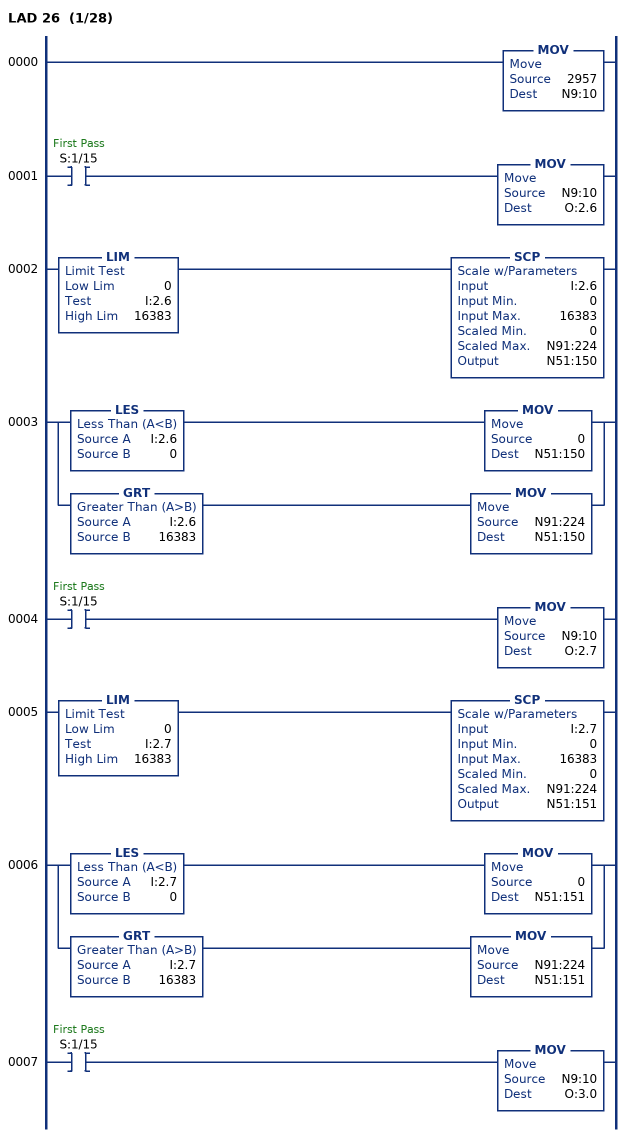
% Rung: 0 %
SOR MOV 2957 N9:10 EOR
% Rung: 1 %
SOR XIC S:1/15 MOV N9:10 O:2.6 EOR
%   S:1/15  "First Pass" %
% Rung: 2 %
SOR LIM 0 I:2.6 16383 SCP I:2.6 0 16383 0 N91:224 N51:150 EOR
% Rung: 3 %
SOR BST LES I:2.6 0 MOV 0 N51:150 NXB GRT I:2.6 16383 MOV N91:224 N51:150 BND EOR
% Rung: 4 %
SOR XIC S:1/15 MOV N9:10 O:2.7 EOR
%   S:1/15  "First Pass" %
% Rung: 5 %
SOR LIM 0 I:2.7 16383 SCP I:2.7 0 16383 0 N91:224 N51:151 EOR
% Rung: 6 %
SOR BST LES I:2.7 0 MOV 0 N51:151 NXB GRT I:2.7 16383 MOV N91:224 N51:151 BND EOR
% Rung: 7 %
SOR XIC S:1/15 MOV N9:10 O:3.0 EOR
%   S:1/15  "First Pass" %

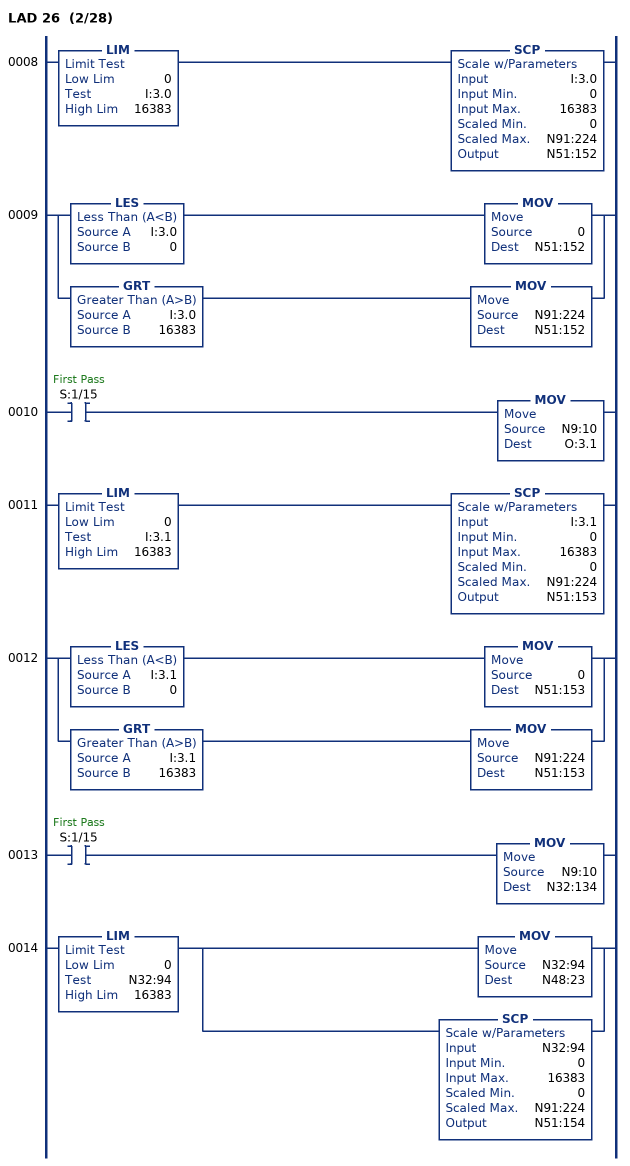
% Rung: 8 %
SOR LIM 0 I:3.0 16383 SCP I:3.0 0 16383 0 N91:224 N51:152 EOR
% Rung: 9 %
SOR BST LES I:3.0 0 MOV 0 N51:152 NXB GRT I:3.0 16383 MOV N91:224 N51:152 BND EOR
% Rung: 10 %
SOR XIC S:1/15 MOV N9:10 O:3.1 EOR
%   S:1/15  "First Pass" %
% Rung: 11 %
SOR LIM 0 I:3.1 16383 SCP I:3.1 0 16383 0 N91:224 N51:153 EOR
% Rung: 12 %
SOR BST LES I:3.1 0 MOV 0 N51:153 NXB GRT I:3.1 16383 MOV N91:224 N51:153 BND EOR
% Rung: 13 %
SOR XIC S:1/15 MOV N9:10 N32:134 EOR
%   S:1/15  "First Pass" %
% Rung: 14 %
SOR LIM 0 N32:94 16383 BST MOV N32:94 N48:23 NXB SCP N32:94 0 16383 0 N91:224 N51:154 BND EOR

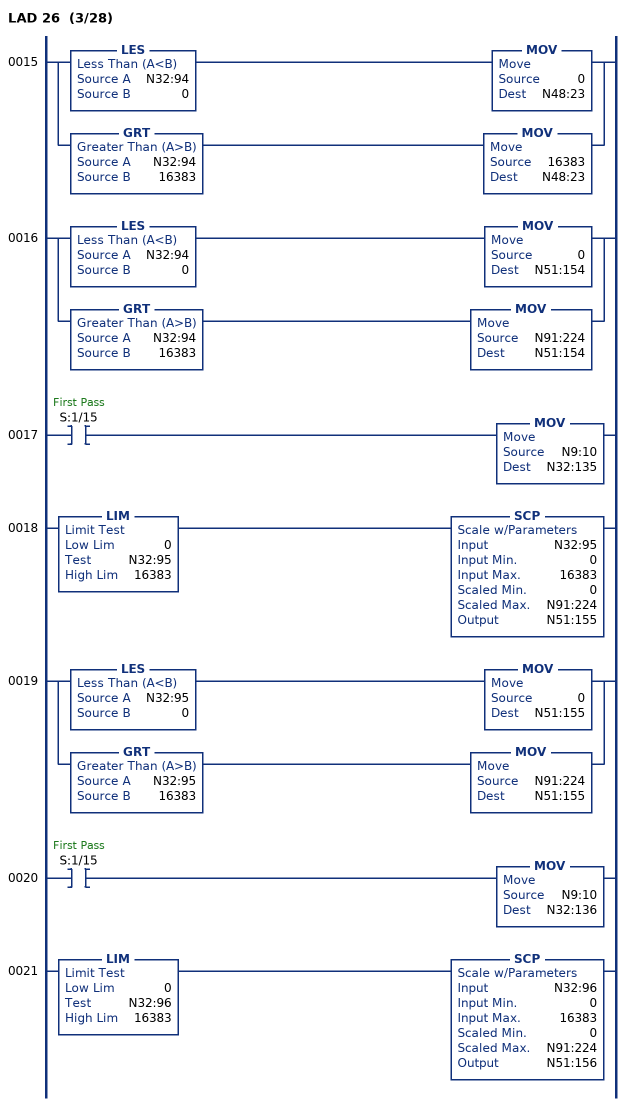
% Rung: 15 %
SOR BST LES N32:94 0 MOV 0 N48:23 NXB GRT N32:94 16383 MOV 16383 N48:23 BND EOR
% Rung: 16 %
SOR BST LES N32:94 0 MOV 0 N51:154 NXB GRT N32:94 16383 MOV N91:224 N51:154 BND EOR
% Rung: 17 %
SOR XIC S:1/15 MOV N9:10 N32:135 EOR
%   S:1/15  "First Pass" %
% Rung: 18 %
SOR LIM 0 N32:95 16383 SCP N32:95 0 16383 0 N91:224 N51:155 EOR
% Rung: 19 %
SOR BST LES N32:95 0 MOV 0 N51:155 NXB GRT N32:95 16383 MOV N91:224 N51:155 BND EOR
% Rung: 20 %
SOR XIC S:1/15 MOV N9:10 N32:136 EOR
%   S:1/15  "First Pass" %
% Rung: 21 %
SOR LIM 0 N32:96 16383 SCP N32:96 0 16383 0 N91:224 N51:156 EOR

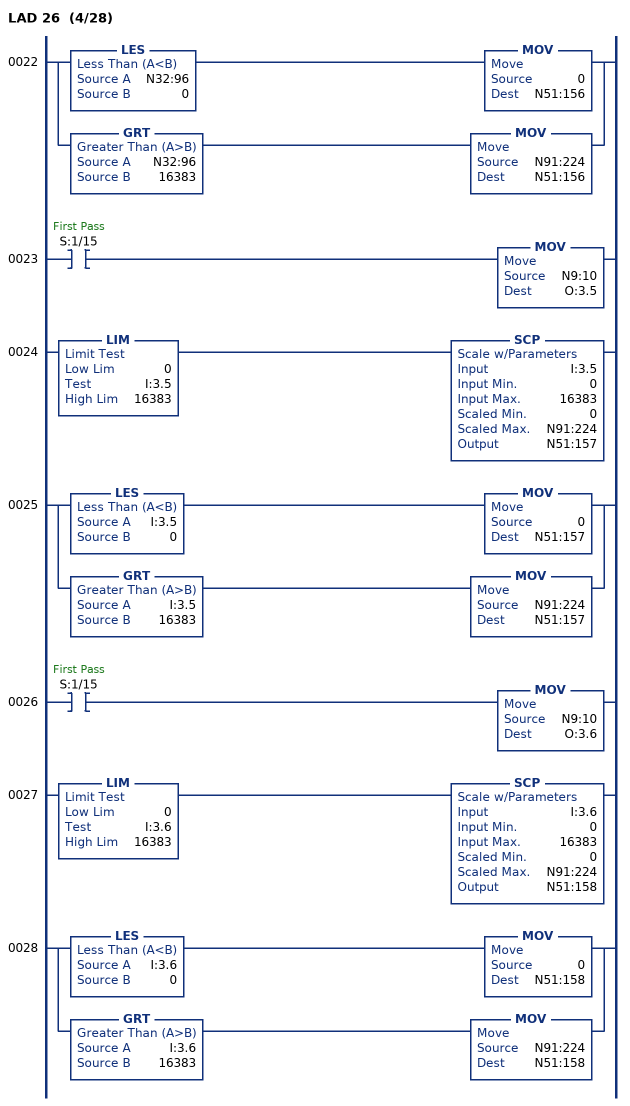
% Rung: 22 %
SOR BST LES N32:96 0 MOV 0 N51:156 NXB GRT N32:96 16383 MOV N91:224 N51:156 BND EOR
% Rung: 23 %
SOR XIC S:1/15 MOV N9:10 O:3.5 EOR
%   S:1/15  "First Pass" %
% Rung: 24 %
SOR LIM 0 I:3.5 16383 SCP I:3.5 0 16383 0 N91:224 N51:157 EOR
% Rung: 25 %
SOR BST LES I:3.5 0 MOV 0 N51:157 NXB GRT I:3.5 16383 MOV N91:224 N51:157 BND EOR
% Rung: 26 %
SOR XIC S:1/15 MOV N9:10 O:3.6 EOR
%   S:1/15  "First Pass" %
% Rung: 27 %
SOR LIM 0 I:3.6 16383 SCP I:3.6 0 16383 0 N91:224 N51:158 EOR
% Rung: 28 %
SOR BST LES I:3.6 0 MOV 0 N51:158 NXB GRT I:3.6 16383 MOV N91:224 N51:158 BND EOR

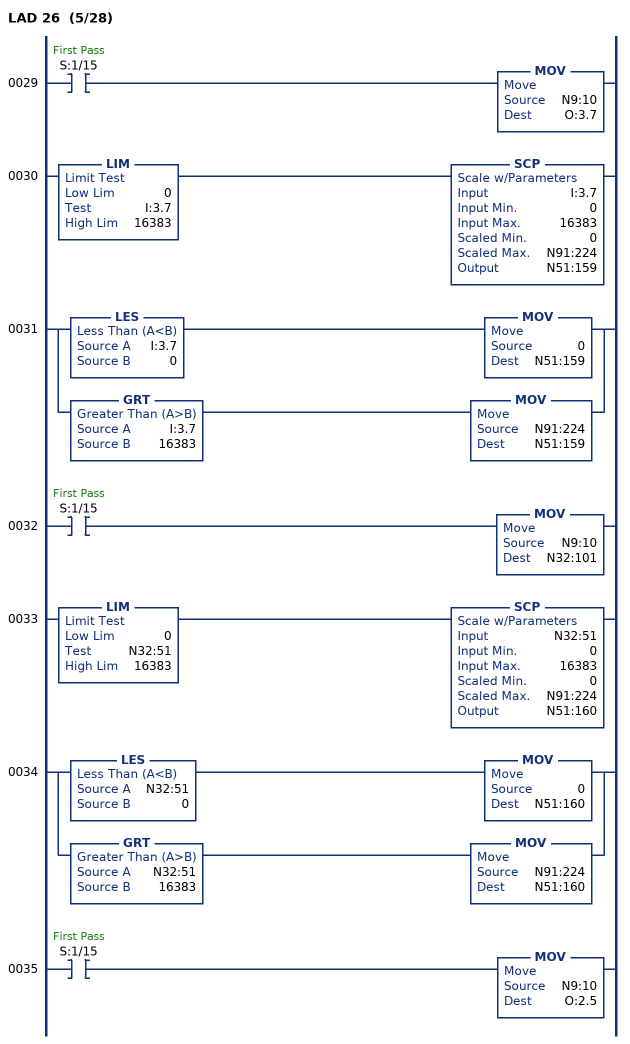
% Rung: 29 %
SOR XIC S:1/15 MOV N9:10 O:3.7 EOR
%   S:1/15  "First Pass" %
% Rung: 30 %
SOR LIM 0 I:3.7 16383 SCP I:3.7 0 16383 0 N91:224 N51:159 EOR
% Rung: 31 %
SOR BST LES I:3.7 0 MOV 0 N51:159 NXB GRT I:3.7 16383 MOV N91:224 N51:159 BND EOR
% Rung: 32 %
SOR XIC S:1/15 MOV N9:10 N32:101 EOR
%   S:1/15  "First Pass" %
% Rung: 33 %
SOR LIM 0 N32:51 16383 SCP N32:51 0 16383 0 N91:224 N51:160 EOR
% Rung: 34 %
SOR BST LES N32:51 0 MOV 0 N51:160 NXB GRT N32:51 16383 MOV N91:224 N51:160 BND EOR
% Rung: 35 %
SOR XIC S:1/15 MOV N9:10 O:2.5 EOR
%   S:1/15  "First Pass" %

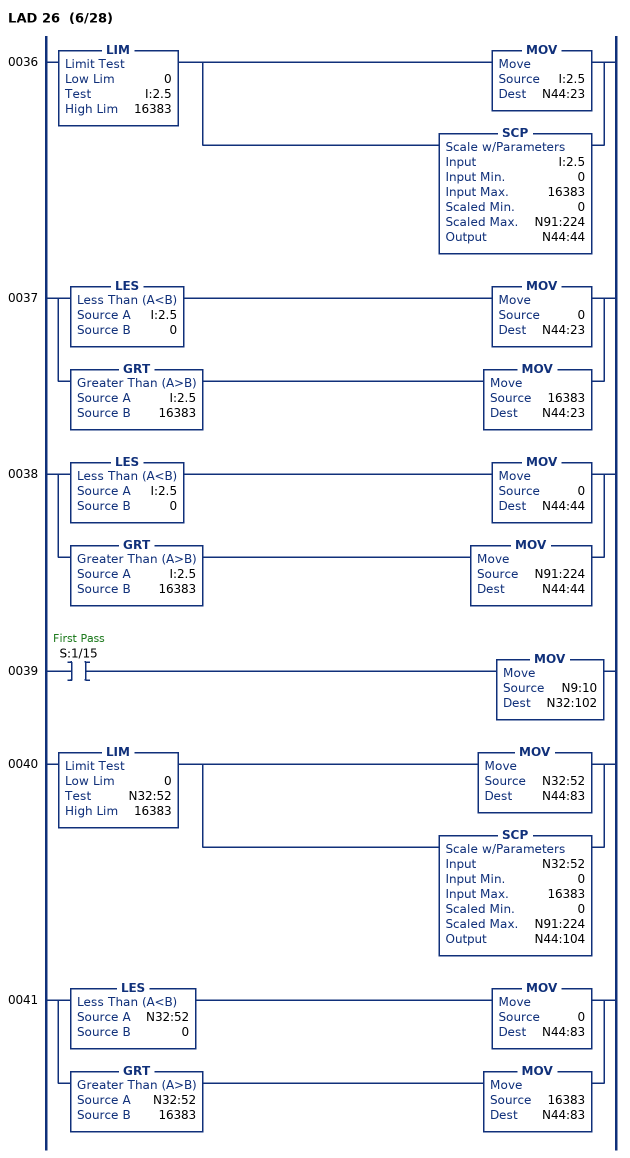
% Rung: 36 %
SOR LIM 0 I:2.5 16383 BST MOV I:2.5 N44:23 NXB SCP I:2.5 0 16383 0 N91:224 N44:44 BND EOR
% Rung: 37 %
SOR BST LES I:2.5 0 MOV 0 N44:23 NXB GRT I:2.5 16383 MOV 16383 N44:23 BND EOR
% Rung: 38 %
SOR BST LES I:2.5 0 MOV 0 N44:44 NXB GRT I:2.5 16383 MOV N91:224 N44:44 BND EOR
% Rung: 39 %
SOR XIC S:1/15 MOV N9:10 N32:102 EOR
%   S:1/15  "First Pass" %
% Rung: 40 %
SOR LIM 0 N32:52 16383 BST MOV N32:52 N44:83 NXB SCP N32:52 0 16383 0 N91:224 N44:104 BND EOR
% Rung: 41 %
SOR BST LES N32:52 0 MOV 0 N44:83 NXB GRT N32:52 16383 MOV 16383 N44:83 BND EOR

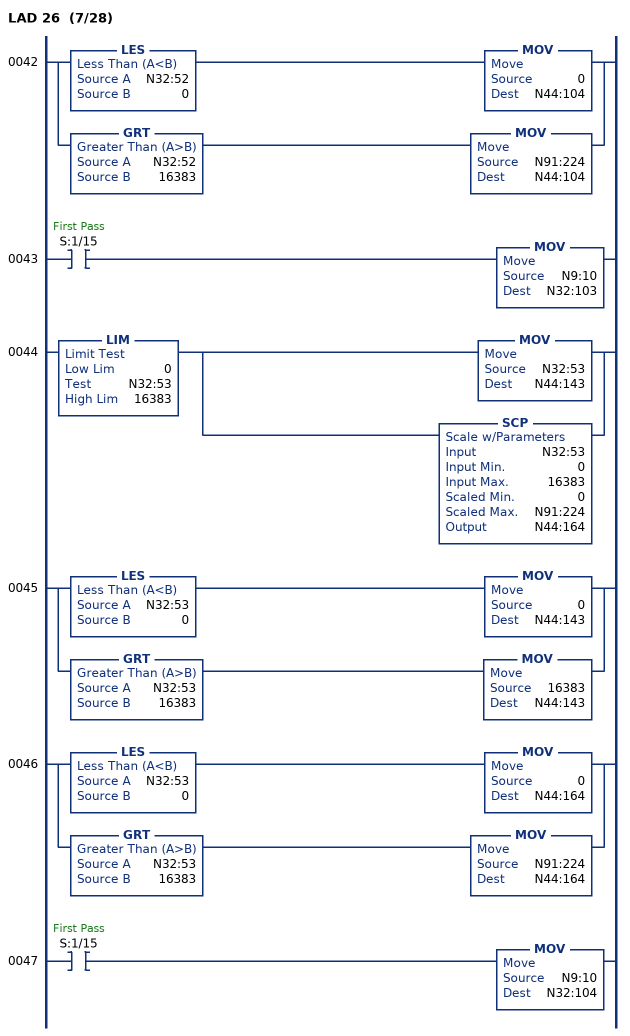
% Rung: 42 %
SOR BST LES N32:52 0 MOV 0 N44:104 NXB GRT N32:52 16383 MOV N91:224 N44:104 BND EOR
% Rung: 43 %
SOR XIC S:1/15 MOV N9:10 N32:103 EOR
%   S:1/15  "First Pass" %
% Rung: 44 %
SOR LIM 0 N32:53 16383 BST MOV N32:53 N44:143 NXB SCP N32:53 0 16383 0 N91:224 N44:164 BND EOR
% Rung: 45 %
SOR BST LES N32:53 0 MOV 0 N44:143 NXB GRT N32:53 16383 MOV 16383 N44:143 BND EOR
% Rung: 46 %
SOR BST LES N32:53 0 MOV 0 N44:164 NXB GRT N32:53 16383 MOV N91:224 N44:164 BND EOR
% Rung: 47 %
SOR XIC S:1/15 MOV N9:10 N32:104 EOR
%   S:1/15  "First Pass" %

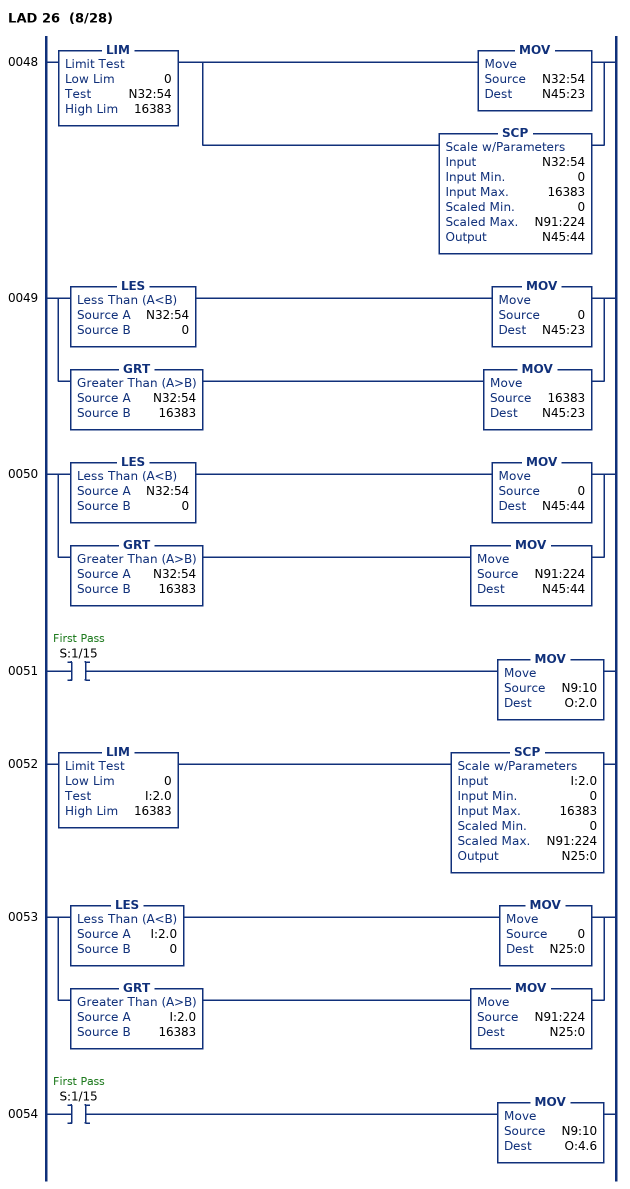
% Rung: 48 %
SOR LIM 0 N32:54 16383 BST MOV N32:54 N45:23 NXB SCP N32:54 0 16383 0 N91:224 N45:44 BND EOR
% Rung: 49 %
SOR BST LES N32:54 0 MOV 0 N45:23 NXB GRT N32:54 16383 MOV 16383 N45:23 BND EOR
% Rung: 50 %
SOR BST LES N32:54 0 MOV 0 N45:44 NXB GRT N32:54 16383 MOV N91:224 N45:44 BND EOR
% Rung: 51 %
SOR XIC S:1/15 MOV N9:10 O:2.0 EOR
%   S:1/15  "First Pass" %
% Rung: 52 %
SOR LIM 0 I:2.0 16383 SCP I:2.0 0 16383 0 N91:224 N25:0 EOR
% Rung: 53 %
SOR BST LES I:2.0 0 MOV 0 N25:0 NXB GRT I:2.0 16383 MOV N91:224 N25:0 BND EOR
% Rung: 54 %
SOR XIC S:1/15 MOV N9:10 O:4.6 EOR
%   S:1/15  "First Pass" %

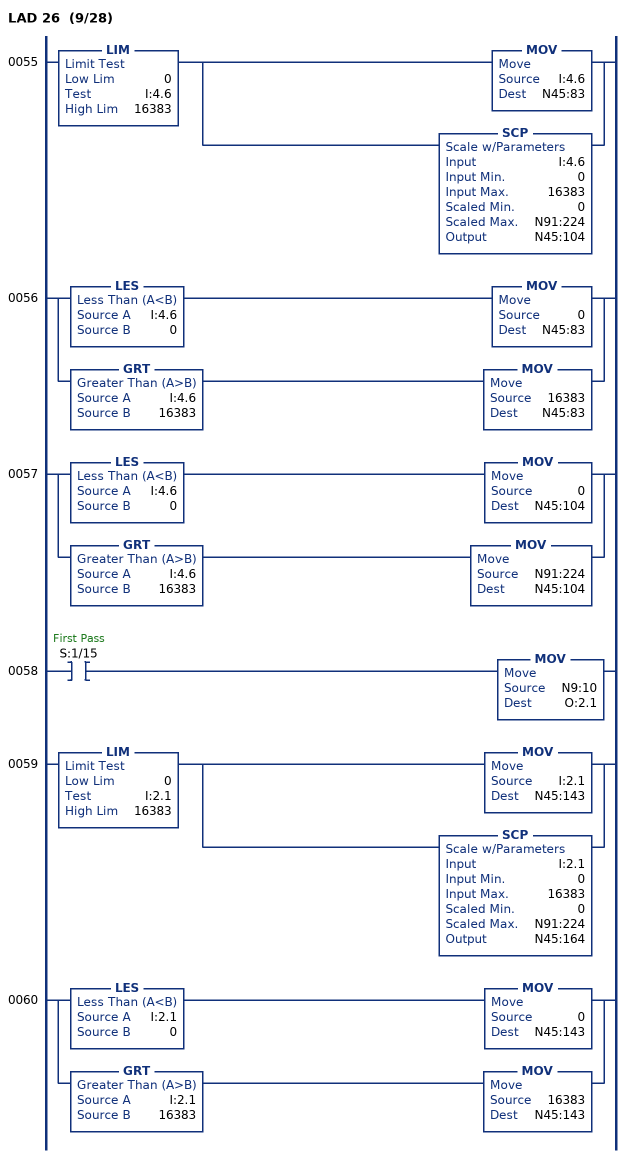
% Rung: 55 %
SOR LIM 0 I:4.6 16383 BST MOV I:4.6 N45:83 NXB SCP I:4.6 0 16383 0 N91:224 N45:104 BND EOR
% Rung: 56 %
SOR BST LES I:4.6 0 MOV 0 N45:83 NXB GRT I:4.6 16383 MOV 16383 N45:83 BND EOR
% Rung: 57 %
SOR BST LES I:4.6 0 MOV 0 N45:104 NXB GRT I:4.6 16383 MOV N91:224 N45:104 BND EOR
% Rung: 58 %
SOR XIC S:1/15 MOV N9:10 O:2.1 EOR
%   S:1/15  "First Pass" %
% Rung: 59 %
SOR LIM 0 I:2.1 16383 BST MOV I:2.1 N45:143 NXB SCP I:2.1 0 16383 0 N91:224 N45:164 BND EOR
% Rung: 60 %
SOR BST LES I:2.1 0 MOV 0 N45:143 NXB GRT I:2.1 16383 MOV 16383 N45:143 BND EOR

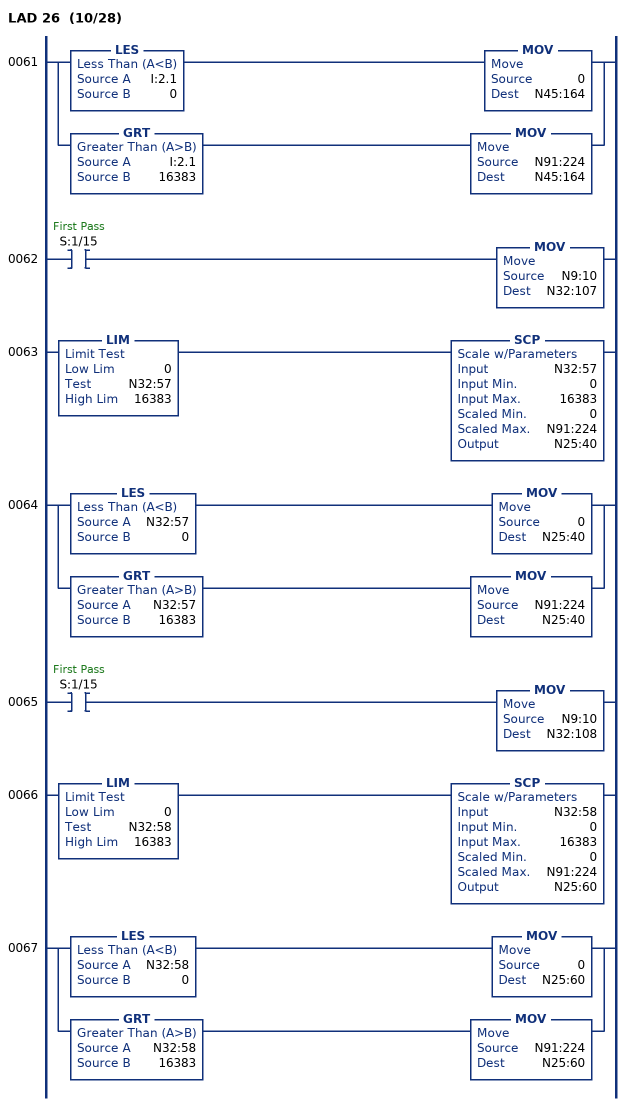
% Rung: 61 %
SOR BST LES I:2.1 0 MOV 0 N45:164 NXB GRT I:2.1 16383 MOV N91:224 N45:164 BND EOR
% Rung: 62 %
SOR XIC S:1/15 MOV N9:10 N32:107 EOR
%   S:1/15  "First Pass" %
% Rung: 63 %
SOR LIM 0 N32:57 16383 SCP N32:57 0 16383 0 N91:224 N25:40 EOR
% Rung: 64 %
SOR BST LES N32:57 0 MOV 0 N25:40 NXB GRT N32:57 16383 MOV N91:224 N25:40 BND EOR
% Rung: 65 %
SOR XIC S:1/15 MOV N9:10 N32:108 EOR
%   S:1/15  "First Pass" %
% Rung: 66 %
SOR LIM 0 N32:58 16383 SCP N32:58 0 16383 0 N91:224 N25:60 EOR
% Rung: 67 %
SOR BST LES N32:58 0 MOV 0 N25:60 NXB GRT N32:58 16383 MOV N91:224 N25:60 BND EOR

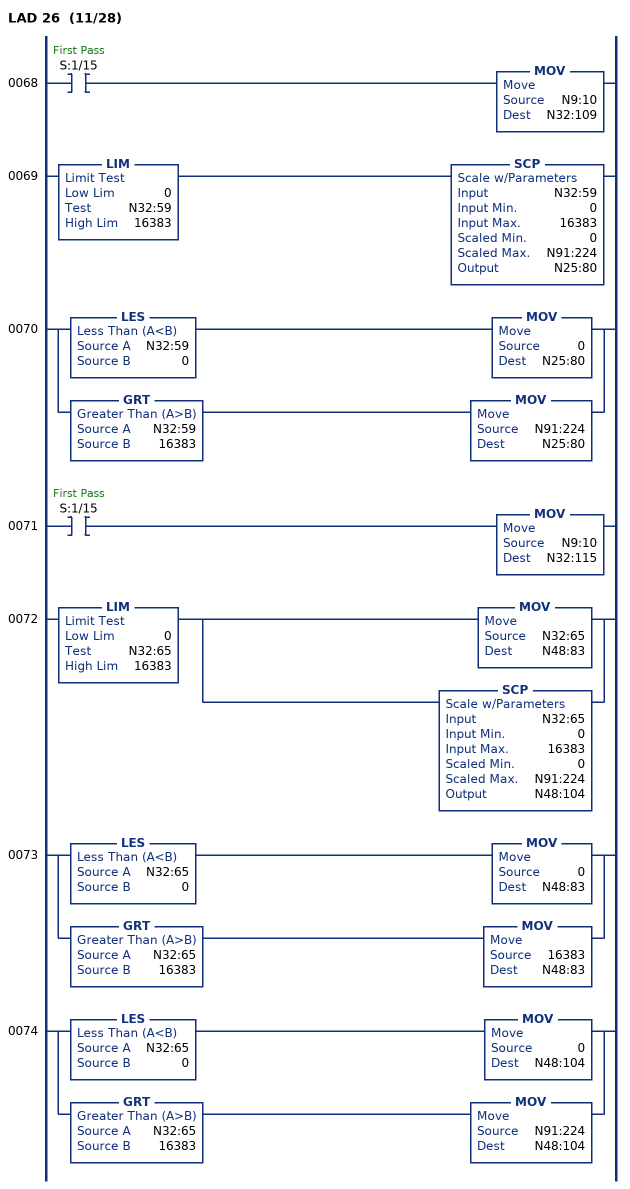
% Rung: 68 %
SOR XIC S:1/15 MOV N9:10 N32:109 EOR
%   S:1/15  "First Pass" %
% Rung: 69 %
SOR LIM 0 N32:59 16383 SCP N32:59 0 16383 0 N91:224 N25:80 EOR
% Rung: 70 %
SOR BST LES N32:59 0 MOV 0 N25:80 NXB GRT N32:59 16383 MOV N91:224 N25:80 BND EOR
% Rung: 71 %
SOR XIC S:1/15 MOV N9:10 N32:115 EOR
%   S:1/15  "First Pass" %
% Rung: 72 %
SOR LIM 0 N32:65 16383 BST MOV N32:65 N48:83 NXB SCP N32:65 0 16383 0 N91:224 N48:104 BND EOR
% Rung: 73 %
SOR BST LES N32:65 0 MOV 0 N48:83 NXB GRT N32:65 16383 MOV 16383 N48:83 BND EOR
% Rung: 74 %
SOR BST LES N32:65 0 MOV 0 N48:104 NXB GRT N32:65 16383 MOV N91:224 N48:104 BND EOR

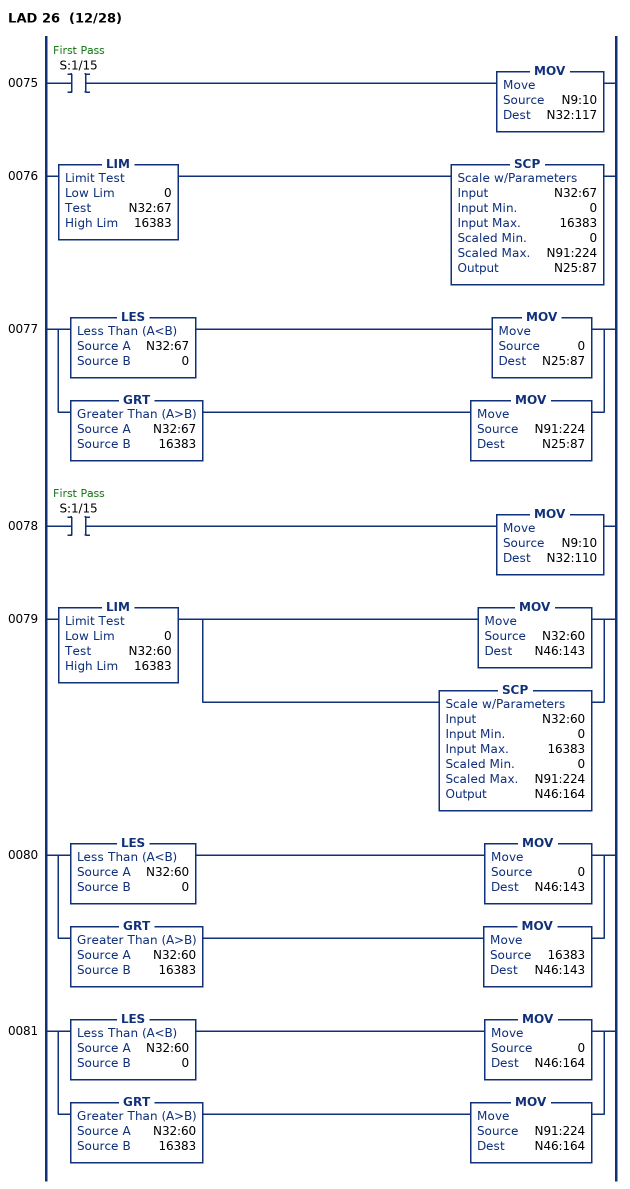
% Rung: 75 %
SOR XIC S:1/15 MOV N9:10 N32:117 EOR
%   S:1/15  "First Pass" %
% Rung: 76 %
SOR LIM 0 N32:67 16383 SCP N32:67 0 16383 0 N91:224 N25:87 EOR
% Rung: 77 %
SOR BST LES N32:67 0 MOV 0 N25:87 NXB GRT N32:67 16383 MOV N91:224 N25:87 BND EOR
% Rung: 78 %
SOR XIC S:1/15 MOV N9:10 N32:110 EOR
%   S:1/15  "First Pass" %
% Rung: 79 %
SOR LIM 0 N32:60 16383 BST MOV N32:60 N46:143 NXB SCP N32:60 0 16383 0 N91:224 N46:164 BND EOR
% Rung: 80 %
SOR BST LES N32:60 0 MOV 0 N46:143 NXB GRT N32:60 16383 MOV 16383 N46:143 BND EOR
% Rung: 81 %
SOR BST LES N32:60 0 MOV 0 N46:164 NXB GRT N32:60 16383 MOV N91:224 N46:164 BND EOR

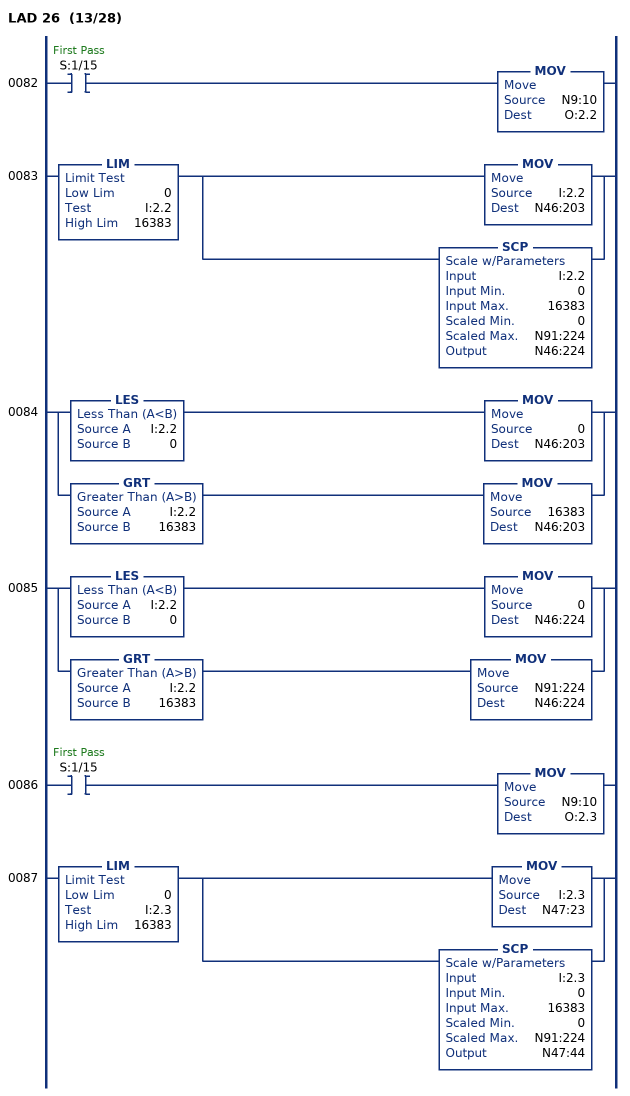
% Rung: 82 %
SOR XIC S:1/15 MOV N9:10 O:2.2 EOR
%   S:1/15  "First Pass" %
% Rung: 83 %
SOR LIM 0 I:2.2 16383 BST MOV I:2.2 N46:203 NXB SCP I:2.2 0 16383 0 N91:224 N46:224 BND EOR
% Rung: 84 %
SOR BST LES I:2.2 0 MOV 0 N46:203 NXB GRT I:2.2 16383 MOV 16383 N46:203 BND EOR
% Rung: 85 %
SOR BST LES I:2.2 0 MOV 0 N46:224 NXB GRT I:2.2 16383 MOV N91:224 N46:224 BND EOR
% Rung: 86 %
SOR XIC S:1/15 MOV N9:10 O:2.3 EOR
%   S:1/15  "First Pass" %
% Rung: 87 %
SOR LIM 0 I:2.3 16383 BST MOV I:2.3 N47:23 NXB SCP I:2.3 0 16383 0 N91:224 N47:44 BND EOR

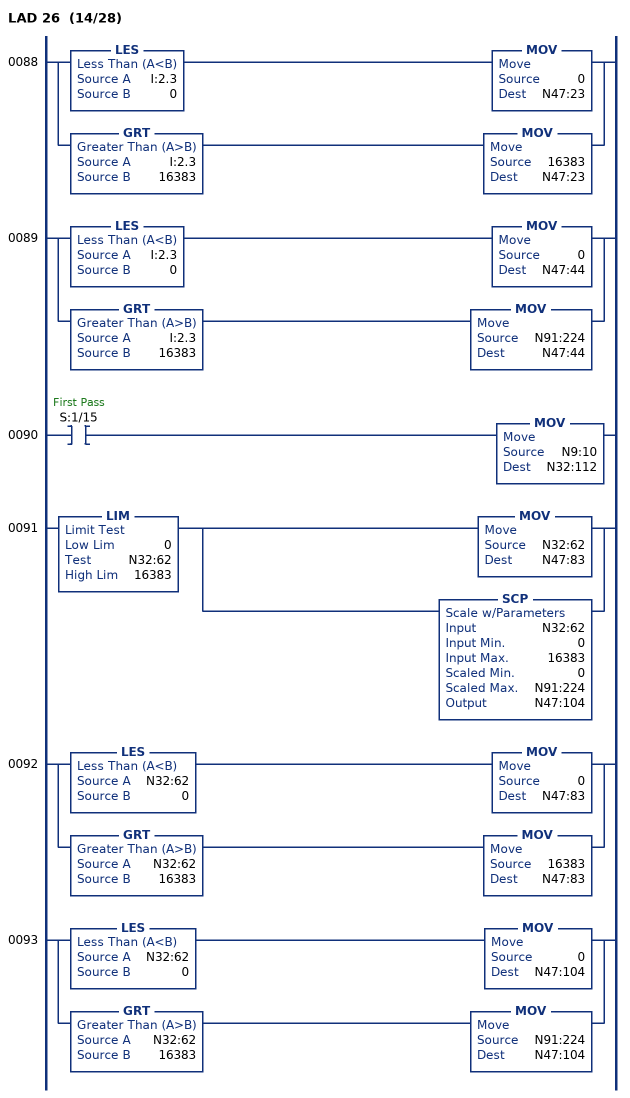
% Rung: 88 %
SOR BST LES I:2.3 0 MOV 0 N47:23 NXB GRT I:2.3 16383 MOV 16383 N47:23 BND EOR
% Rung: 89 %
SOR BST LES I:2.3 0 MOV 0 N47:44 NXB GRT I:2.3 16383 MOV N91:224 N47:44 BND EOR
% Rung: 90 %
SOR XIC S:1/15 MOV N9:10 N32:112 EOR
%   S:1/15  "First Pass" %
% Rung: 91 %
SOR LIM 0 N32:62 16383 BST MOV N32:62 N47:83 NXB SCP N32:62 0 16383 0 N91:224 N47:104 BND EOR
% Rung: 92 %
SOR BST LES N32:62 0 MOV 0 N47:83 NXB GRT N32:62 16383 MOV 16383 N47:83 BND EOR
% Rung: 93 %
SOR BST LES N32:62 0 MOV 0 N47:104 NXB GRT N32:62 16383 MOV N91:224 N47:104 BND EOR

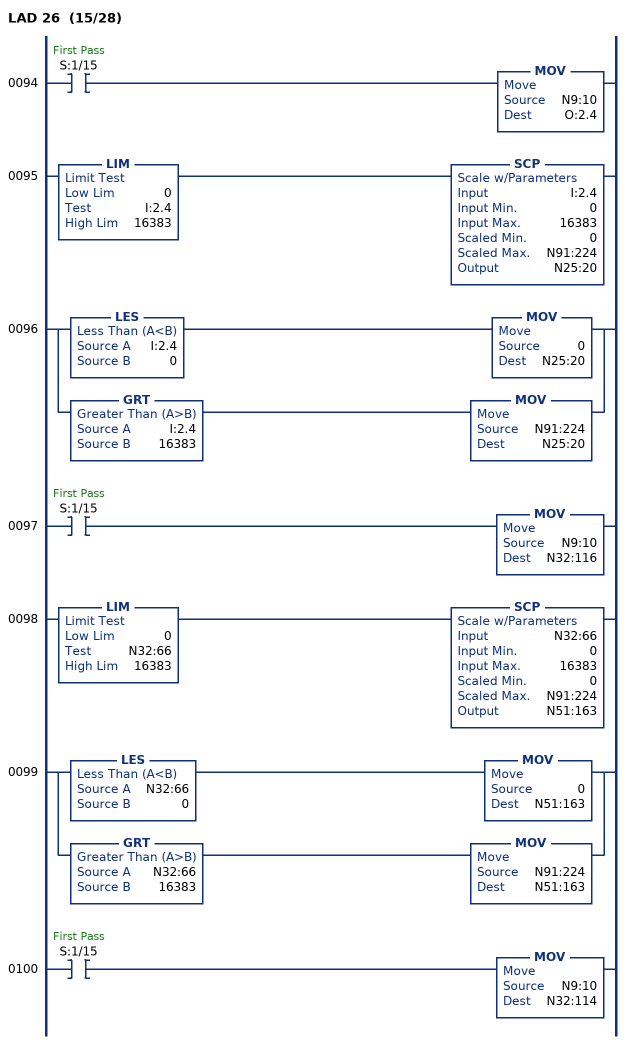
% Rung: 94 %
SOR XIC S:1/15 MOV N9:10 O:2.4 EOR
%   S:1/15  "First Pass" %
% Rung: 95 %
SOR LIM 0 I:2.4 16383 SCP I:2.4 0 16383 0 N91:224 N25:20 EOR
% Rung: 96 %
SOR BST LES I:2.4 0 MOV 0 N25:20 NXB GRT I:2.4 16383 MOV N91:224 N25:20 BND EOR
% Rung: 97 %
SOR XIC S:1/15 MOV N9:10 N32:116 EOR
%   S:1/15  "First Pass" %
% Rung: 98 %
SOR LIM 0 N32:66 16383 SCP N32:66 0 16383 0 N91:224 N51:163 EOR
% Rung: 99 %
SOR BST LES N32:66 0 MOV 0 N51:163 NXB GRT N32:66 16383 MOV N91:224 N51:163 BND EOR
% Rung: 100 %
SOR XIC S:1/15 MOV N9:10 N32:114 EOR
%   S:1/15  "First Pass" %

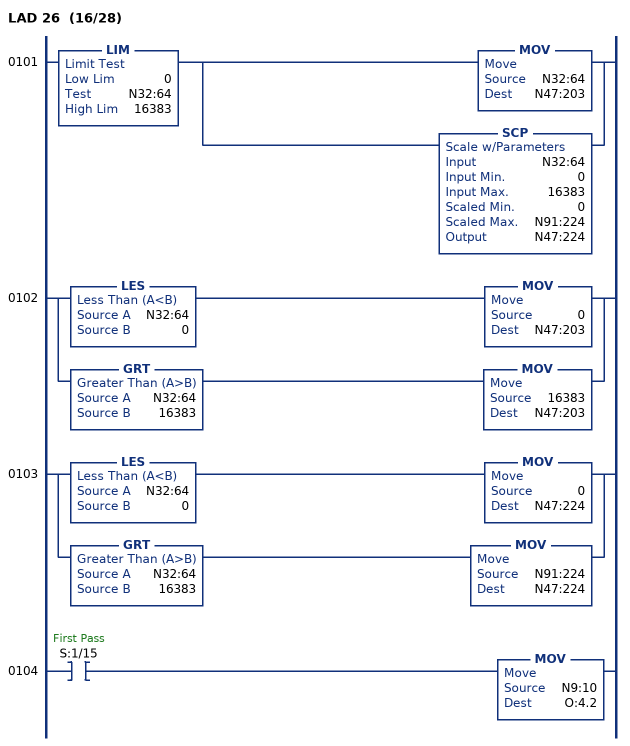
% Rung: 101 %
SOR LIM 0 N32:64 16383 BST MOV N32:64 N47:203 NXB SCP N32:64 0 16383 0 N91:224 N47:224 BND EOR
% Rung: 102 %
SOR BST LES N32:64 0 MOV 0 N47:203 NXB GRT N32:64 16383 MOV 16383 N47:203 BND EOR
% Rung: 103 %
SOR BST LES N32:64 0 MOV 0 N47:224 NXB GRT N32:64 16383 MOV N91:224 N47:224 BND EOR
% Rung: 104 %
SOR XIC S:1/15 MOV N9:10 O:4.2 EOR
%   S:1/15  "First Pass" %

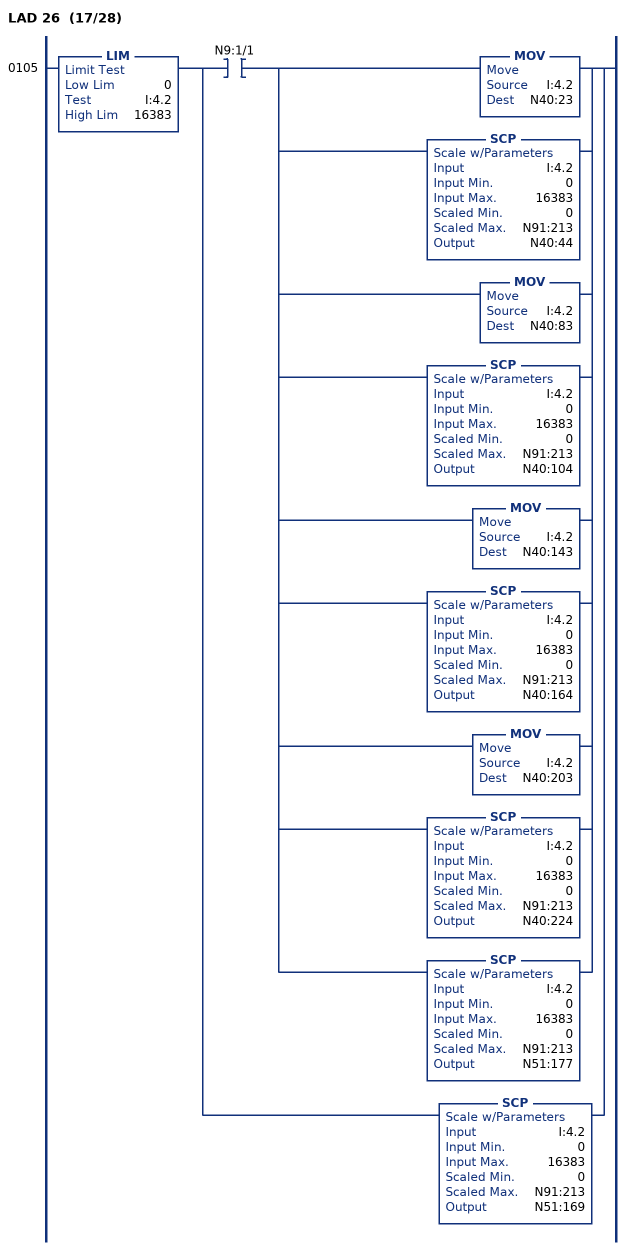
% Rung: 105 %
SOR LIM 0 I:4.2 16383 BST XIC N9:1/1 BST MOV I:4.2 N40:23 NXB SCP I:4.2 0 16383 0 N91:213 N40:44 NXB MOV I:4.2 N40:83 NXB SCP I:4.2 0 16383 0 N91:213 N40:104 NXB MOV I:4.2 N40:143 NXB SCP I:4.2 0 16383 0 N91:213 N40:164 NXB MOV I:4.2 N40:203 NXB SCP I:4.2 0 16383 0 N91:213 N40:224 NXB SCP I:4.2 0 16383 0 N91:213 N51:177 BND NXB SCP I:4.2 0 16383 0 N91:213 N51:169 BND EOR

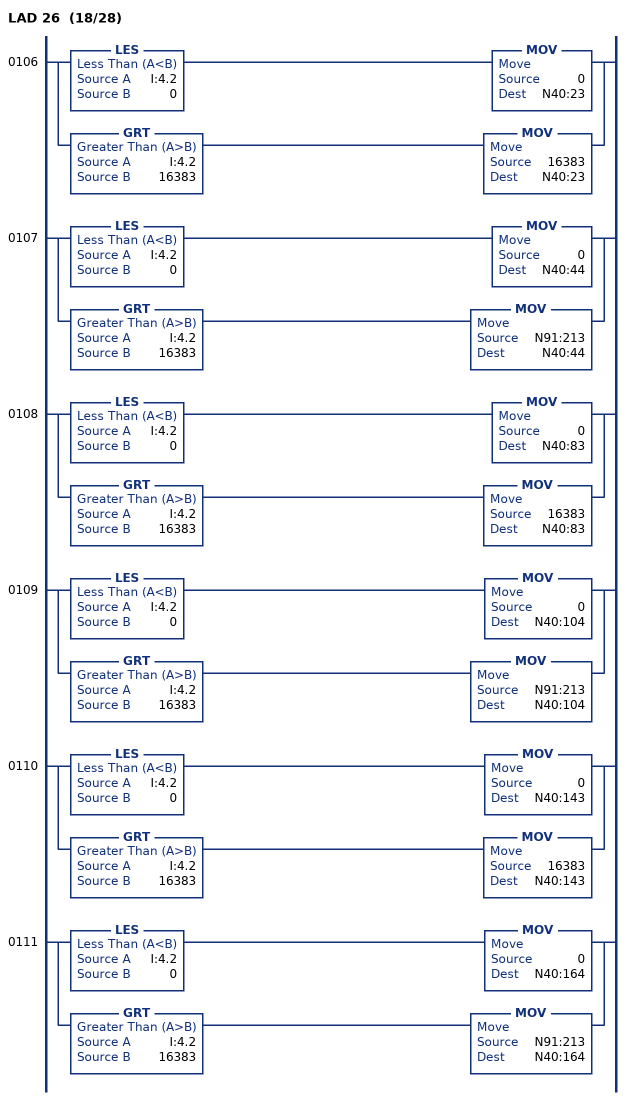
% Rung: 106 %
SOR BST LES I:4.2 0 MOV 0 N40:23 NXB GRT I:4.2 16383 MOV 16383 N40:23 BND EOR
% Rung: 107 %
SOR BST LES I:4.2 0 MOV 0 N40:44 NXB GRT I:4.2 16383 MOV N91:213 N40:44 BND EOR
% Rung: 108 %
SOR BST LES I:4.2 0 MOV 0 N40:83 NXB GRT I:4.2 16383 MOV 16383 N40:83 BND EOR
% Rung: 109 %
SOR BST LES I:4.2 0 MOV 0 N40:104 NXB GRT I:4.2 16383 MOV N91:213 N40:104 BND EOR
% Rung: 110 %
SOR BST LES I:4.2 0 MOV 0 N40:143 NXB GRT I:4.2 16383 MOV 16383 N40:143 BND EOR
% Rung: 111 %
SOR BST LES I:4.2 0 MOV 0 N40:164 NXB GRT I:4.2 16383 MOV N91:213 N40:164 BND EOR

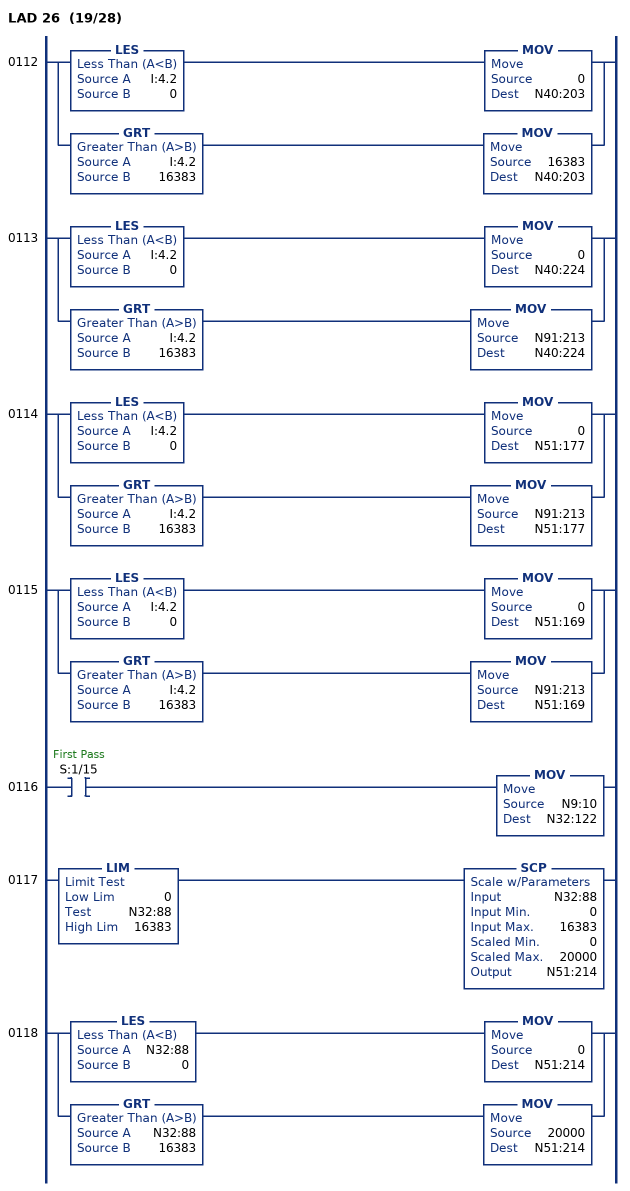
% Rung: 112 %
SOR BST LES I:4.2 0 MOV 0 N40:203 NXB GRT I:4.2 16383 MOV 16383 N40:203 BND EOR
% Rung: 113 %
SOR BST LES I:4.2 0 MOV 0 N40:224 NXB GRT I:4.2 16383 MOV N91:213 N40:224 BND EOR
% Rung: 114 %
SOR BST LES I:4.2 0 MOV 0 N51:177 NXB GRT I:4.2 16383 MOV N91:213 N51:177 BND EOR
% Rung: 115 %
SOR BST LES I:4.2 0 MOV 0 N51:169 NXB GRT I:4.2 16383 MOV N91:213 N51:169 BND EOR
% Rung: 116 %
SOR XIC S:1/15 MOV N9:10 N32:122 EOR
%   S:1/15  "First Pass" %
% Rung: 117 %
SOR LIM 0 N32:88 16383 SCP N32:88 0 16383 0 20000 N51:214 EOR
% Rung: 118 %
SOR BST LES N32:88 0 MOV 0 N51:214 NXB GRT N32:88 16383 MOV 20000 N51:214 BND EOR

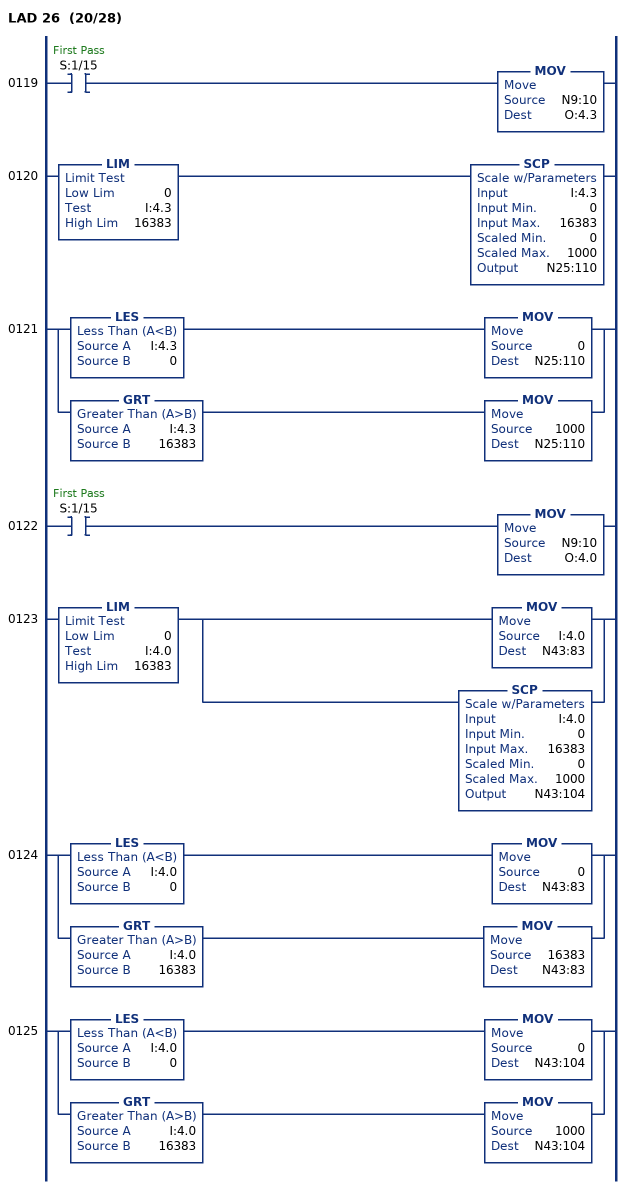
% Rung: 119 %
SOR XIC S:1/15 MOV N9:10 O:4.3 EOR
%   S:1/15  "First Pass" %
% Rung: 120 %
SOR LIM 0 I:4.3 16383 SCP I:4.3 0 16383 0 1000 N25:110 EOR
% Rung: 121 %
SOR BST LES I:4.3 0 MOV 0 N25:110 NXB GRT I:4.3 16383 MOV 1000 N25:110 BND EOR
% Rung: 122 %
SOR XIC S:1/15 MOV N9:10 O:4.0 EOR
%   S:1/15  "First Pass" %
% Rung: 123 %
SOR LIM 0 I:4.0 16383 BST MOV I:4.0 N43:83 NXB SCP I:4.0 0 16383 0 1000 N43:104 BND EOR
% Rung: 124 %
SOR BST LES I:4.0 0 MOV 0 N43:83 NXB GRT I:4.0 16383 MOV 16383 N43:83 BND EOR
% Rung: 125 %
SOR BST LES I:4.0 0 MOV 0 N43:104 NXB GRT I:4.0 16383 MOV 1000 N43:104 BND EOR

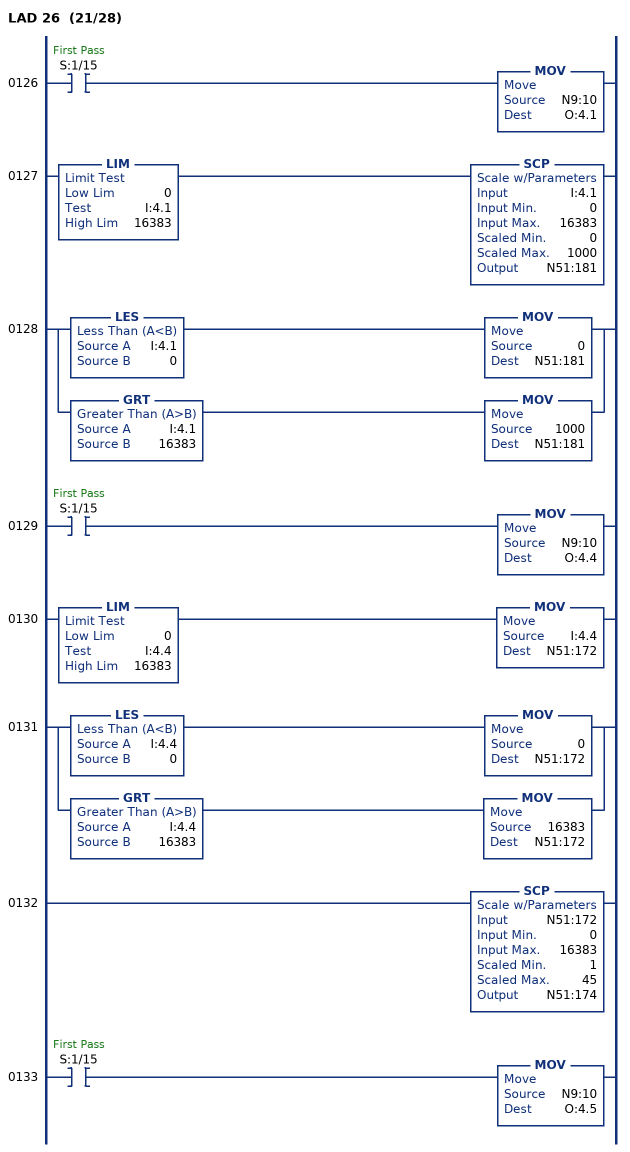
% Rung: 126 %
SOR XIC S:1/15 MOV N9:10 O:4.1 EOR
%   S:1/15  "First Pass" %
% Rung: 127 %
SOR LIM 0 I:4.1 16383 SCP I:4.1 0 16383 0 1000 N51:181 EOR
% Rung: 128 %
SOR BST LES I:4.1 0 MOV 0 N51:181 NXB GRT I:4.1 16383 MOV 1000 N51:181 BND EOR
% Rung: 129 %
SOR XIC S:1/15 MOV N9:10 O:4.4 EOR
%   S:1/15  "First Pass" %
% Rung: 130 %
SOR LIM 0 I:4.4 16383 MOV I:4.4 N51:172 EOR
% Rung: 131 %
SOR BST LES I:4.4 0 MOV 0 N51:172 NXB GRT I:4.4 16383 MOV 16383 N51:172 BND EOR
% Rung: 132 %
SOR SCP N51:172 0 16383 1 45 N51:174 EOR
% Rung: 133 %
SOR XIC S:1/15 MOV N9:10 O:4.5 EOR
%   S:1/15  "First Pass" %

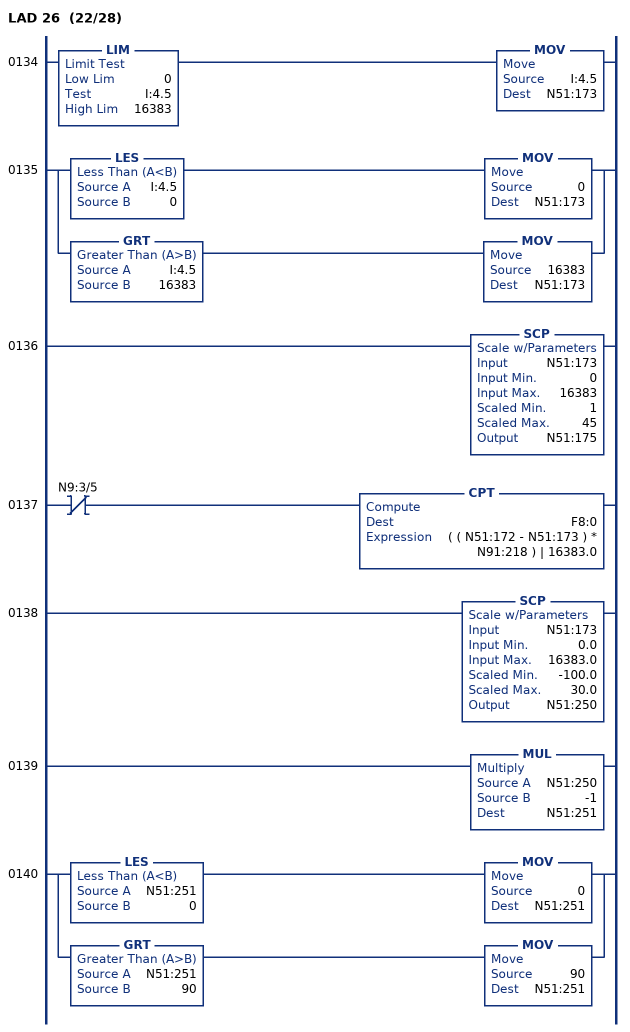
% Rung: 134 %
SOR LIM 0 I:4.5 16383 MOV I:4.5 N51:173 EOR
% Rung: 135 %
SOR BST LES I:4.5 0 MOV 0 N51:173 NXB GRT I:4.5 16383 MOV 16383 N51:173 BND EOR
% Rung: 136 %
SOR SCP N51:173 0 16383 1 45 N51:175 EOR
% Rung: 137 %
SOR XIO N9:3/5 CPT F8:0 " ( ( N51:172 - N51:173 ) * N91:218 ) | 16383.0 " EOR
% Rung: 138 %
SOR SCP N51:173 0.0 16383.0 -100.0 30.0 N51:250 EOR
% Rung: 139 %
SOR MUL N51:250 -1 N51:251 EOR
% Rung: 140 %
SOR BST LES N51:251 0 MOV 0 N51:251 NXB GRT N51:251 90 MOV 90 N51:251 BND EOR

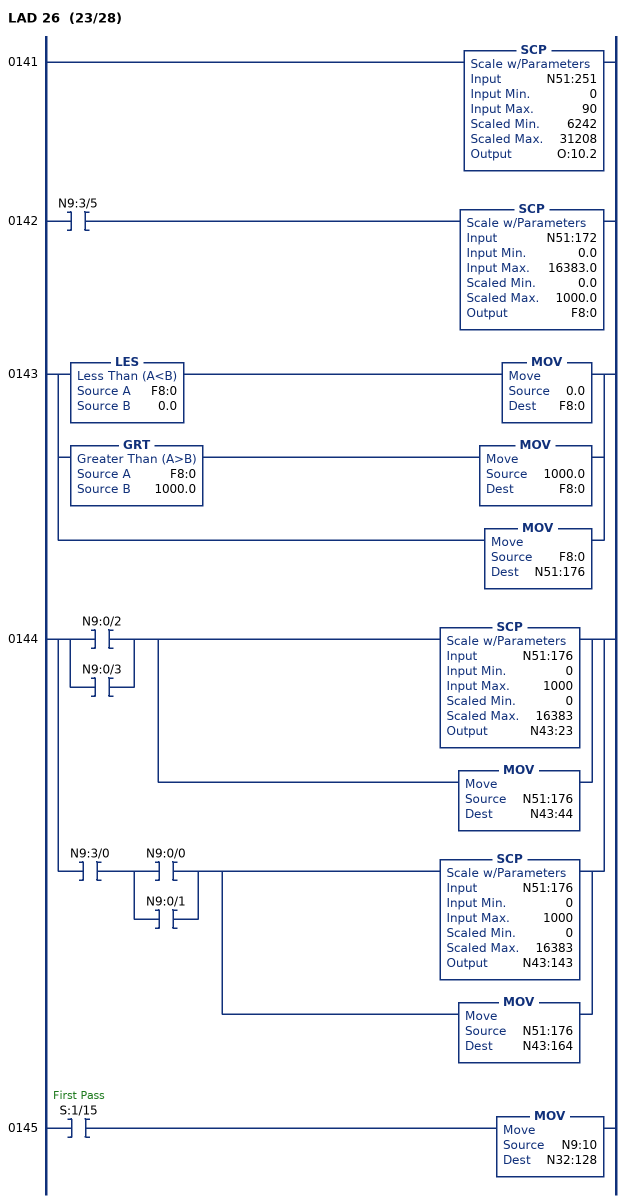
% Rung: 141 %
SOR SCP N51:251 0 90 6242 31208 O:10.2 EOR
% Rung: 142 %
SOR XIC N9:3/5 SCP N51:172 0.0 16383.0 0.0 1000.0 F8:0 EOR
% Rung: 143 %
SOR BST LES F8:0 0.0 MOV 0.0 F8:0 NXB GRT F8:0 1000.0 MOV 1000.0 F8:0 NXB MOV F8:0 N51:176 BND EOR
% Rung: 144 %
SOR BST BST XIC N9:0/2 NXB XIC N9:0/3 BND BST SCP N51:176 0 1000 0 16383 N43:23 NXB MOV N51:176 N43:44 BND NXB XIC N9:3/0 BST XIC N9:0/0 NXB XIC N9:0/1 BND BST SCP N51:176 0 1000 0 16383 N43:143 NXB MOV N51:176 N43:164 BND BND EOR
% Rung: 145 %
SOR XIC S:1/15 MOV N9:10 N32:128 EOR
%   S:1/15  "First Pass" %

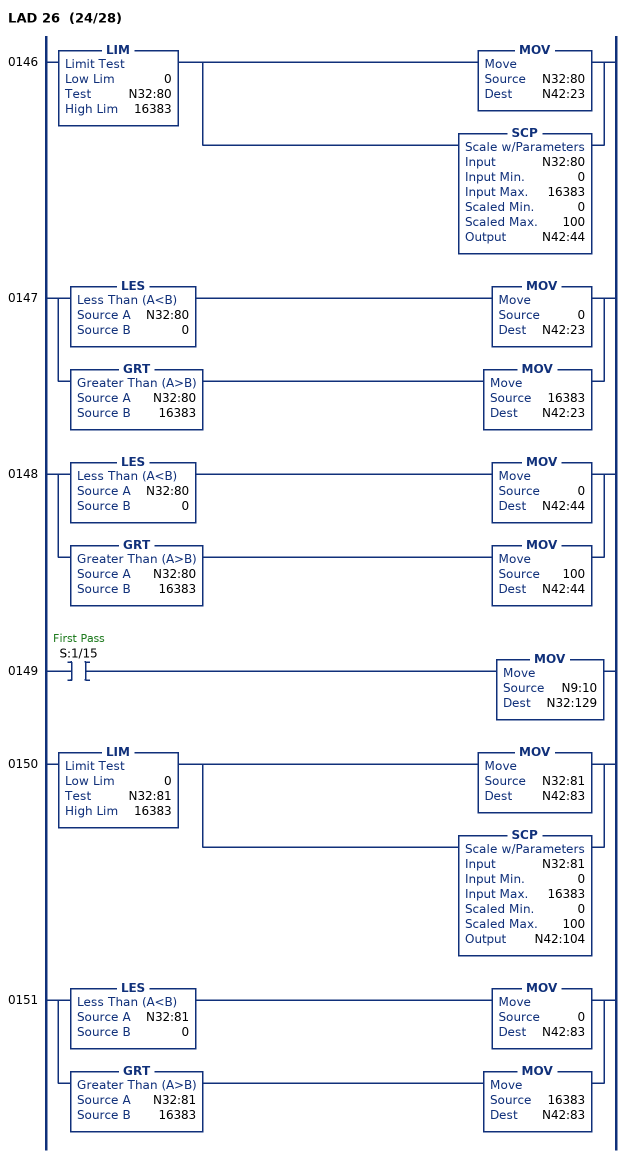
% Rung: 146 %
SOR LIM 0 N32:80 16383 BST MOV N32:80 N42:23 NXB SCP N32:80 0 16383 0 100 N42:44 BND EOR
% Rung: 147 %
SOR BST LES N32:80 0 MOV 0 N42:23 NXB GRT N32:80 16383 MOV 16383 N42:23 BND EOR
% Rung: 148 %
SOR BST LES N32:80 0 MOV 0 N42:44 NXB GRT N32:80 16383 MOV 100 N42:44 BND EOR
% Rung: 149 %
SOR XIC S:1/15 MOV N9:10 N32:129 EOR
%   S:1/15  "First Pass" %
% Rung: 150 %
SOR LIM 0 N32:81 16383 BST MOV N32:81 N42:83 NXB SCP N32:81 0 16383 0 100 N42:104 BND EOR
% Rung: 151 %
SOR BST LES N32:81 0 MOV 0 N42:83 NXB GRT N32:81 16383 MOV 16383 N42:83 BND EOR

